	        //Set Signaling Request
	        IF #R_TRIG_PreStartSemiAutomaticUp.Q OR #R_TRIG_PreStartSemiAutomaticDown.Q THEN
	            #iqUDT_EquipmentControl.Request.SignalingRequest := TRUE;
	        END_IF;

	        IF #sx_SemiAutomatic
	            AND (NOT #ix_PRXUp
	            AND #sx_UpRequest)
	            OR #sUDT_HMIStatus.Specific.SwitchingTimerError
	        THEN
	            #sx_UpRequest := false;
	            #sx_PreStartSemiAutomaticUp := false;
	        END_IF;

	        IF #sx_SemiAutomatic
	            AND (NOT #ix_PRXDown
	            AND #sx_DownRequest)
	            OR #sUDT_HMIStatus.Specific.SwitchingTimerError
	        THEN
	            #sx_DownRequest := false;
	            #sx_PreStartSemiAutomaticDown := false;
	        END_IF;

	    END_REGION

	    REGION 7.2 - Start/Stop AB switch conveyor directly

	        // Start
	        IF #iqUDT_EquipmentControl.Command.Start                                       // Start from system
	            AND #sx_Ready                                                               // Equipment has no errors
	        THEN
	            #qx_ExternalHold := FALSE;                                           // External stop signal
	        END_IF;

	        // Stop
	        IF #sUDT_HMIStatus.Specific.UpperSwitchAreaError                                // Blockage of switching area
	            OR #sUDT_HMIStatus.Specific.LowerSwitchAreaError
	            OR NOT #sx_SemiAutomatic                                                    // The AB switch is not (semi-)automatic active
	        THEN
	            #qx_ExternalHold := TRUE;                                            // External stop signal
	        END_IF;

	    END_REGION

	END_REGION

	REGION 8 - Write interface DB signals

	    REGION 8.1 - Signal interface

	        #iqUDT_ABSwitchInterface.InternalErrorReset := #iqUDT_EquipmentControl.Command.Reset;      // Write Reset signal to the VFD interface
	        #iqUDT_ABSwitchInterface.ResetStatistics := #iqUDT_EquipmentControl.Command.ResetData;     // Write Reset data signal to the VFD interface

	    END_REGION

	    REGION 8.1 - Mode selection

	        #ss_ABSwitch_Interface.SemiAutomatic :=
	        (#sx_SemiAutomatic                                                               // Automatic started
	        OR #sx_Stopping);                                                                // stopping is activated Go to default position

	        #ss_ABSwitch_Interface.Manual :=
	        #ix_SSMan                                                             // Manual mode is started
	        AND (#sx_CombinedJogUp                                                           // IF selected jog in positive direction
	        OR #sx_CombinedJogDown);

	    END_REGION

	    REGION 8.2 - Run enable

	        #ss_ABSwitch_Interface.RunEnabled :=                                                  // Enable the positioning device to run
	        NOT #iqUDT_ABSwitchInterface.InternalErrorVFD                               // or there are errors in the VFD
	        AND NOT #sx_ConfigurationError                                                   // configuration is wrong
	        AND #ix_HardwareOk                                                        // or an internal error in the RIO panel occured
	        AND (#ss_ABSwitch_Interface.SemiAutomatic                                             // AB switch is in semi-automatic mode
	        OR (#ss_ABSwitch_Interface.Manual                                                     // manual mode is active
	        AND (#sx_CombinedJogUp                                                           // If selected jog in positive direction
	        OR #sx_CombinedJogDown)));                                                       // If selected jog in negative direction

	    END_REGION

	END_REGION

	REGION 9 - Positions reached

	    // triggers of PEC's down/up
	    #F_TRIG_PECUp(CLK := #ix_PRXUp);
	    #F_TRIG_PECDown(CLK := #ix_PRXDown);

	    // when the upper photo eye to stop the AB switch is covered it means the position is reached
	    IF #F_TRIG_PECUp.Q THEN
	        #sx_UpperPositionReached := true;
	    ELSIF #sx_DownRequest OR #ix_SSMan THEN
	        #sx_UpperPositionReached := false;
	    END_IF;

	    // when the lower photo eye to stop the AB switch is covered it means the position is reached
	    IF #F_TRIG_PECDown.Q THEN
	        #sx_LowerPositionReached := true;
	    ELSIF #sx_UpRequest OR #ix_SSMan THEN
	        #sx_LowerPositionReached := false;
	    END_IF;

	END_REGION

	REGION 10 - Run up/down

	    // Conditions to run AB switch down
	    #iqUDT_ABSwitchInterface.RunRvs := ((#sx_DownRequest AND #sx_SemiAutomatic)
	    OR #sx_JogDown)
	    AND NOT #sx_LowerPositionReached
	    AND #ss_ABSwitch_Interface.RunEnabled
	    AND #ix_PRXDown
	    AND NOT #sUDT_HMIStatus.Specific.LimitSensorLowerPosition;

	    // Conditions to run AB switch upwards
	    #iqUDT_ABSwitchInterface.RunFwd := ((#sx_UpRequest AND #sx_SemiAutomatic)
	    OR #sx_JogUp)
	    AND NOT #sx_UpperPositionReached
	    AND #ss_ABSwitch_Interface.RunEnabled
	    AND #ix_PRXUp
	    AND NOT #sUDT_HMIStatus.Specific.LimitSensorUpperPosition;

	END_REGION

	REGION 11 - AB switch speed reduction

	    #F_TRIG_PECBrakeUp(CLK := #ix_PRXBrkUp);

	    #F_TRIG_PECBrakeDown(CLK := #ix_PRXBrkDwn);

	    IF #F_TRIG_PECBrakeUp.Q
	        AND #iqUDT_ABSwitchInterface.RunFwd
	    THEN
	        #sx_ABSwitchSlowSpeedUp := TRUE;
	    END_IF;

	    IF #F_TRIG_PECBrakeDown.Q
	        AND #iqUDT_ABSwitchInterface.RunRvs
	    THEN
	        #sx_ABSwitchSlowSpeedDown := TRUE;
	    END_IF;

	    IF ((#ss_ABSwitch_Interface.Positioning
	        AND #iqUDT_ABSwitchInterface.RunFwd
	        AND #sx_ABSwitchSlowSpeedUp
	        AND #ix_PRXUp)
	        OR
	        (#ss_ABSwitch_Interface.Positioning
	        AND #iqUDT_ABSwitchInterface.RunRvs
	        AND #sx_ABSwitchSlowSpeedDown
	        AND #ix_PRXDown))
	    THEN
	        #iqUDT_ABSwitchInterface.SpeedSetpoint := #iUDT_ABSwitchConfig.BrakingSpeedSetpoint;
	    ELSE
	        #iqUDT_ABSwitchInterface.SpeedSetpoint := #iUDT_ABSwitchConfig.NominalSpeedSetPoint;
	        #sx_ABSwitchSlowSpeedUp := FALSE;
	        #sx_ABSwitchSlowSpeedDown := FALSE;
	    END_IF;

	    IF #ss_ABSwitch_Interface.Manual THEN
	        #iqUDT_ABSwitchInterface.SpeedSetpoint := #iUDT_ABSwitchConfig.ManualModeSpeed;
	    END_IF;

	END_REGION

	REGION 12 - Statistics

	    // Down Time
	    IF #sx_SemiAutomatic                                                                 // Automatic active
	        AND NOT #sx_Ready                                                                // Conveyor not ready
	        OR #iqUDT_EquipmentControl.Command.ResetData                                    // Reset statistics
	    THEN

	        "FC_Statistics"(ix_Reset := #iqUDT_EquipmentControl.Command.ResetData,              // Or reset statistics from control
	                        ix_Activate := #sx_SemiAutomatic AND NOT #sx_Ready,                     // AB switch is stopped
	                        ix_RTrigActivate := #R_TRIG_DownTime.Q,                                      // AB switch is stopped triger
	                        iqUDT_Statistics := #iqUDT_Statistics.DownTime);                            // AB switch is stopped statistics
	    END_IF;

	    // Up time
	    IF #sx_SemiAutomatic                                // Automatic active
	        AND #sx_Ready                                   // Ready active
	        OR #iqUDT_EquipmentControl.Command.ResetData   // Reset statistics
	    THEN
	        "FC_Statistics"(ix_Reset := #iqUDT_EquipmentControl.Command.ResetData,        // OR reset statistics from control
	                        ix_Activate := #sx_SemiAutomatic AND #sx_Ready,                   // AB switch is running
	                        ix_RTrigActivate := #R_TRIG_UpTime.Q,                                  // AB switch running trigger
	                        iqUDT_Statistics := #iqUDT_Statistics.UpTime);                        // AB switch running statistics

	    END_IF;

	    // Upper switch area error
	    #R_TRIG_UPSwA_Error(CLK := #sUDT_HMIStatus.Specific.UpperSwitchAreaError);               // Oneshot trigger error occurred

	    IF #iqUDT_ABSwitchInterface.ResetStatistics OR                                         // IF there is signal TO reset statistics from AB switch interface
	        #iqUDT_EquipmentControl.Command.ResetData OR                                        // Or there is signal to reset statistics from equipment control structure
	        #sUDT_HMIStatus.Specific.UpperSwitchAreaError                                        // Or an upper switch area error occurred
	    THEN

	        "FC_Statistics"(ix_Reset := #iqUDT_ABSwitchInterface.ResetStatistics OR                 // Reset statistics from HMI
	                        #iqUDT_EquipmentControl.Command.ResetData,                                       // Or reset statistics from control
	                        ix_Activate := #sUDT_HMIStatus.Specific.UpperSwitchAreaError,               // Upper switch area error occurred
	                        ix_RTrigActivate := #R_TRIG_UPSwA_Error.Q,                                       // Error trigger
	                        iqUDT_Statistics := #iqUDT_Statistics.UpperSwitchArea_Error);                   // Statistics of AB switch errors

	    END_IF;

	    // Lower switch area error
	    #R_TRIG_LowSwA_Error(CLK := #sUDT_HMIStatus.Specific.LowerSwitchAreaError);              // Oneshot trigger error occurred

	    IF #iqUDT_ABSwitchInterface.ResetStatistics OR                                          // IF there is signal TO reset statistics from AB switch interface
	        #iqUDT_EquipmentControl.Command.ResetData OR                                        // Or there is signal to reset statistics from equipment control structure
	        #sUDT_HMIStatus.Specific.LowerSwitchAreaError                                        // Or an upper switch area error occurred
	    THEN

	        "FC_Statistics"(ix_Reset := #iqUDT_ABSwitchInterface.ResetStatistics OR                 // Reset statistics from HMI
	                        #iqUDT_EquipmentControl.Command.ResetData,                                       // Or reset statistics from control
	                        ix_Activate := #sUDT_HMIStatus.Specific.LowerSwitchAreaError,               // Upper switch area error occurred
	                        ix_RTrigActivate := #R_TRIG_LowSwA_Error.Q,                                      // Error trigger
	                        iqUDT_Statistics := #iqUDT_Statistics.LowerSwitchArea_Error);                   // Statistics of AB switch errors

	    END_IF;

	END_REGION

	REGION 13 - Status

	    #sUDT_Status.Stopped := #sx_Ready AND NOT #sx_SemiAutomatic AND NOT #sx_Stopping;      // stopped
	    #sUDT_Status.AutoON := #sx_SemiAutomatic OR #sx_Stopping;                              // Auto On
	    #sUDT_Status.Halted := FALSE;                                                          // Halted
	    #sUDT_Status.Dieback := FALSE;                                                         // Die back
	    #sUDT_Status.Running := (#sx_UpRequest OR #sx_DownRequest) AND #sx_SemiAutomatic;      // Running
	    #sUDT_Status.ManualRun := #ix_SSMan AND #sUDT_Status.Running;              // Manual run
	    #sUDT_Status.Manual := #ix_SSMan;                                           // Manual
	    #sUDT_Status.EnergySave := FALSE;                                                      // Energy save active
	    #sUDT_Status.SafetyStop := NOT #ix_SafetyOk;                                           // Safety not ok

	    IF #sUDT_StatusOld <> #sUDT_Status                                            // update on change
	    THEN

	        // Set status to status number
	        #sUDT_HMIStatus.Status := 0;                                               // Initialise status number

	        IF #sUDT_Status.Running                                                    // Running
	        THEN

	            #sUDT_HMIStatus.Status := "DB_HMIStatusConfiguration".Running;

	        END_IF;

	        IF #sUDT_Status.Stopped                                                    // Stopped
	        THEN

	            #sUDT_HMIStatus.Status := "DB_HMIStatusConfiguration".Stopped;

	        END_IF;

	        IF #sUDT_Status.Dieback                                                    // Dieback
	        THEN

	            #sUDT_HMIStatus.Status := "DB_HMIStatusConfiguration".Dieback;

	        END_IF;

	        IF #sUDT_Status.ManualRun                                                  // Manual run
	        THEN

	            #sUDT_HMIStatus.Status := "DB_HMIStatusConfiguration".ManualRun;

	        END_IF;

	        IF #sUDT_Status.Manual                                                     // Manual
	        THEN

	            #sUDT_HMIStatus.Status := "DB_HMIStatusConfiguration".Manual;

	        END_IF;

	        IF #iqUDT_ABSwitchInterface.InternalWarningVFD                                  // The VFD has an internal warning
	            OR NOT #ix_HardwareOk                                                         // The RIO panel has an internal warning

	        THEN

	            #sUDT_HMIStatus.Status := "DB_HMIStatusConfiguration".Warning;

	        END_IF;

	        IF #sUDT_HMIStatus.Specific.UpperSwitchAreaError                           // Upper limit switch error
	            OR #sUDT_HMIStatus.Specific.LowerSwitchAreaError                       // Lower limit switch error
	        THEN

	            #sUDT_HMIStatus.Status := "DB_HMIStatusConfiguration".VFDError;

	        END_IF;

	        IF #iqUDT_ABSwitchInterface.InternalErrorVFD                                // The VFD has an internal error
	            OR NOT #ix_HardwareOk                                                    // The RIO panel has an internal error
	        THEN

	            #sUDT_HMIStatus.Status := "DB_HMIStatusConfiguration".Error;

	        END_IF;


	        IF #sUDT_Status.SafetyStop                                                 // Safety stop
	        THEN

	            #sUDT_HMIStatus.Status := "DB_HMIStatusConfiguration".SafetyStop;

	        END_IF;

	        // Copy status to output
	        #sUDT_StatusOld := #sUDT_Status;                                          // Copy status TO memory
	        #qUDT_Status := #sUDT_Status;                                             // Copy status to output

	    END_IF;

	    //   Specific status
	    #sUDT_HMIStatus.Specific.UpperPosition := #sx_ActualPositionUP;
	    #sUDT_HMIStatus.Specific.LowerPosition := #sx_ActualPositionDown;

	    #qUDT_HMIStatus := #sUDT_HMIStatus;

	END_REGION

	REGION 14 - Report to control block

	    "FC_EquipmentReport"(iUDT_Status := #sUDT_Status,
	                         iqUDT_Control := #iqUDT_EquipmentControl);

	END_REGION

	REGION 15 - Internal errors and warnings reset

	    #iqUDT_ABSwitchInterface.InternalErrorPEC := FALSE;
	    #iqUDT_ABSwitchInterface.InternalWarningTracking := FALSE;
	    #iqUDT_ABSwitchInterface.InternalErrorTracking := FALSE;
	    #iqUDT_ABSwitchInterface.InternalWarningVFD := FALSE;
	    #iqUDT_ABSwitchInterface.InternalErrorVFD := FALSE;
	    #iqUDT_ABSwitchInterface.Disconnected := FALSE;

	END_REGION

END_FUNCTION_BLOCK

